SYSTEM Project_499
  (* Version 1.0, 2024-12-17, Bruno *)
  APPLICATION Project_499App
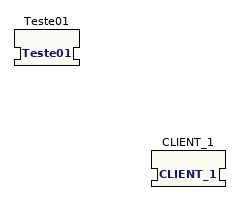
    FBS
      Teste01 : Teste01;
      CLIENT_1 : CLIENT_1;
    END_FBS
  END_APPLICATION
END_SYSTEM
